{attribute 'qualified_only'}
{attribute 'strict'}
TYPE E_STATE :
(
	normal := 0,
	error := 1
);
END_TYPE

(* stored: Version 1.1.0.1, ProductVersion 3.1.4024.12
   DUT E_STATE: Id {7c14b72c-c073-496b-a718-29433bc8d6e5} *)
